FUNCTION rt_floord : LREAL
VAR_INPUT
	u: LREAL;
END_VAR
VAR
END_VAR


rt_floord := DINT_TO_LREAL(TRUNC(u));

IF u = rt_floord THEN 
    rt_floord := u;
ELSIF u < 0.0 THEN 
    rt_floord := rt_floord - 1.0;
END_IF;

END_FUNCTION

(* stored: Version 1.1.0.1, ProductVersion 3.1.4024.12
   POU rt_floord: Id {6b511f2b-646b-4e76-a867-b53887a8a7c0}, SpecialFunc None *)
